Fanuc KAREL source: kb00105.KL

-- PROVISIONAL review KL for V940-1; original PC SHA256 80574ec08348379789e71e410a97d45a35d06e652b08169b852f055fb73a31f4
-- Incomplete behavior may be omitted. Consult companion uncertainty JSON. Do not deploy.
PROGRAM KB00105
%NOLOCKGROUP
BEGIN
  -- V9_ZERO_TABLE_METADATA_HINT layout=0002_ascii; no indexed target words; source/name/runtime held
  -- UNRESOLVED_PC offsets 5-14; opcodes 3F,75
  -- UNRESOLVED_PC offsets 19-28; opcodes 3F,75
  -- UNRESOLVED_PC offsets 33-40; opcodes 9D,23
  -- UNRESOLVED_PC offsets 45-52; opcodes 9D,23
  -- UNRESOLVED_PC offsets 57-64; opcodes 9D,23
  -- UNRESOLVED_PC offsets 69-76; opcodes 9D,23
  -- UNRESOLVED_PC offsets 81-88; opcodes 9D,23
  -- UNRESOLVED_PC offsets 93-100; opcodes 9D,23
  -- UNRESOLVED_PC offsets 105-112; opcodes 9D,23
  -- UNRESOLVED_PC offsets 117-126; opcodes 3F,75
  -- UNRESOLVED_PC offsets 131-138; opcodes 9D,23
  -- UNRESOLVED_PC offsets 143-219; opcodes 27,22,2A,22,2A,22,22,22,22,22,22,22,22,2A,22,31
  -- UNRESOLVED_PC offsets 224-228; opcodes 7F
END KB00105
